PROGRAM TestStationControl
VAR
	(* These timers are used to imitate the moving time in the visualization*)
	T_Mat_Check: TIME := TIME#2S0MS;
	T1: TIME := TIME#2S0MS;
	T_liftDown: TIME := TIME#2S0MS;
	T_H_meas: TIME := TIME#2S0MS;
	T_MatPush: TIME := TIME#1S0MS;
	TON_Mat_Check: TON;
	TON_MatPush: TON;
	TON_MatPush2: TON;
	TON_Lift: TON;
	TON1: TON;
	TON_0: TON;
	TON_1: TON;
	TON_2: TON;
	TON_H_Meas: TON;
	TON_Lift2: TON;
	TON_reset: TON;
	
	(* These are just used to maintain the sequence or flow*)
	next2: BOOL;
	next3: BOOL;
	next4: BOOL;
END_VAR
VAR // added by the converter: edge detectors and wires of the graphical bodies
    _w1, _w2, _w3, _w4, _w5, _w6, _w7 : BOOL;
END_VAR

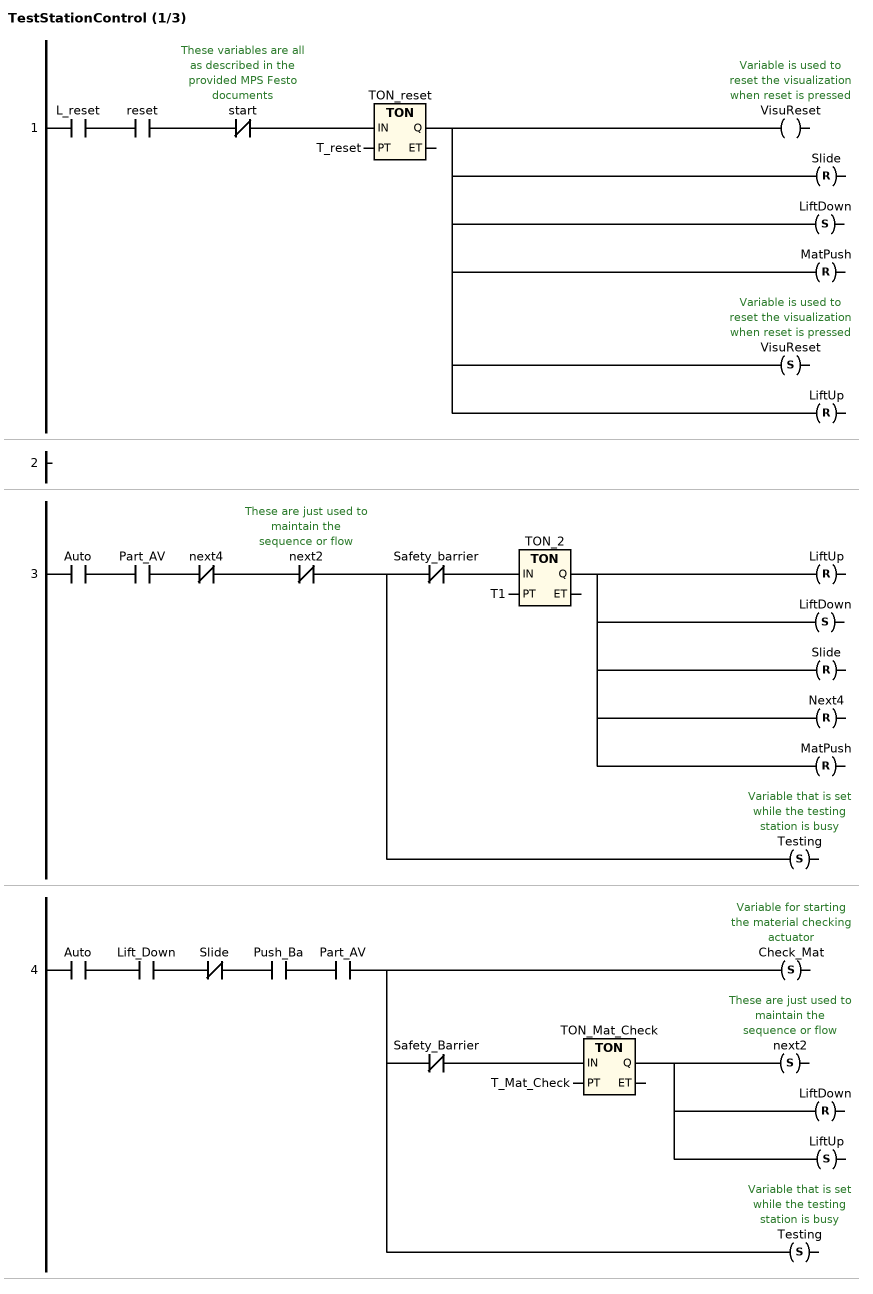
// NETWORK 1
//   start: These variables are all as described in the provided MPS Festo documents
//   T_reset: time to imitate reset value
//   VisuReset: Variable is used to reset the visualization when reset is pressed
TON_reset(IN := L_reset AND reset AND NOT start, PT := T_reset); // TON
VisuReset := TON_reset.Q;
Slide R= TON_reset.Q;
LiftDown S= TON_reset.Q;
MatPush R= TON_reset.Q;
VisuReset S= TON_reset.Q;
LiftUp R= TON_reset.Q;

// NETWORK 2

// NETWORK 3
//   next2: These are just used to maintain the sequence or flow
//   Testing: Variable that is set while the testing station is busy
_w1 := Auto AND Part_AV AND NOT next4 AND NOT next2;
TON_2(IN := _w1 AND NOT Safety_barrier, PT := T1); // TON
LiftUp R= TON_2.Q;
LiftDown S= TON_2.Q;
Slide R= TON_2.Q;
Next4 R= TON_2.Q;
MatPush R= TON_2.Q;
Testing S= _w1;

// NETWORK 4
//   Check_Mat: Variable for starting the material checking actuator
//   T_Mat_Check: These timers are used to imitate the moving time in the visualization
//   next2: These are just used to maintain the sequence or flow
//   Testing: Variable that is set while the testing station is busy
_w2 := Auto AND Lift_Down AND NOT Slide AND Push_Ba AND Part_AV;
Check_Mat S= _w2;
TON_Mat_Check(IN := _w2 AND NOT Safety_Barrier, PT := T_Mat_Check); // TON
next2 S= TON_Mat_Check.Q;
LiftDown R= TON_Mat_Check.Q;
LiftUp S= TON_Mat_Check.Q;
Testing S= _w2;

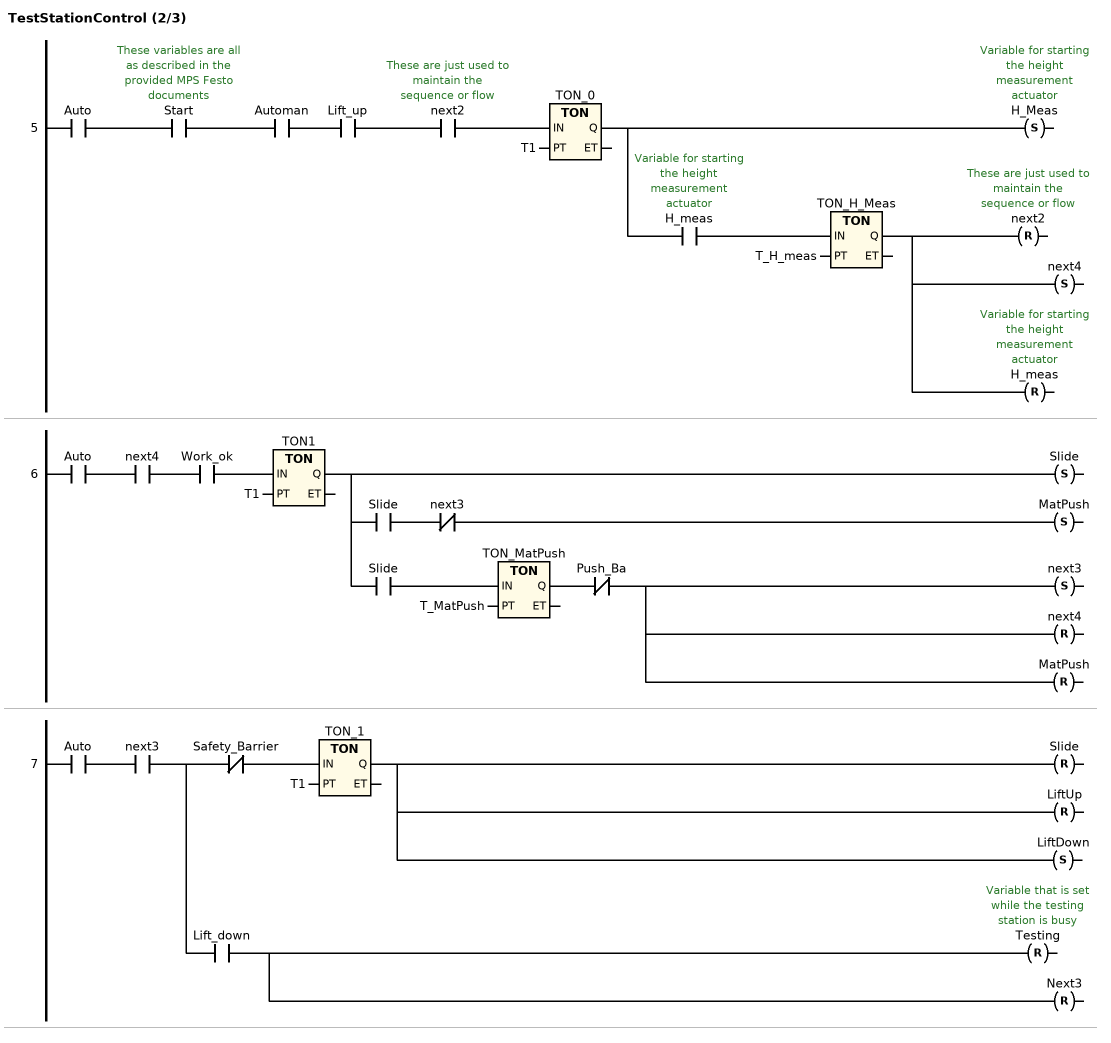
// NETWORK 5
//   Start: These variables are all as described in the provided MPS Festo documents
//   next2: These are just used to maintain the sequence or flow
//   H_Meas: Variable for starting the height measurement actuator
//   H_meas: Variable for starting the height measurement actuator
TON_0(IN := Auto AND Start AND Automan AND Lift_up AND next2, PT := T1); // TON
H_Meas S= TON_0.Q;
TON_H_Meas(IN := TON_0.Q AND H_meas, PT := T_H_meas); // TON
next2 R= TON_H_Meas.Q;
next4 S= TON_H_Meas.Q;
H_meas R= TON_H_Meas.Q;

// NETWORK 6
TON1(IN := Auto AND next4 AND Work_ok, PT := T1); // TON
Slide S= TON1.Q;
MatPush S= TON1.Q AND Slide AND NOT next3;
TON_MatPush(IN := TON1.Q AND Slide, PT := T_MatPush); // TON
_w3 := TON_MatPush.Q AND NOT Push_Ba;
next3 S= _w3;
next4 R= _w3;
MatPush R= _w3;

// NETWORK 7
//   Testing: Variable that is set while the testing station is busy
_w4 := Auto AND next3;
TON_1(IN := _w4 AND NOT Safety_Barrier, PT := T1); // TON
Slide R= TON_1.Q;
LiftUp R= TON_1.Q;
LiftDown S= TON_1.Q;
_w5 := _w4 AND Lift_down;
Testing R= _w5;
Next3 R= _w5;

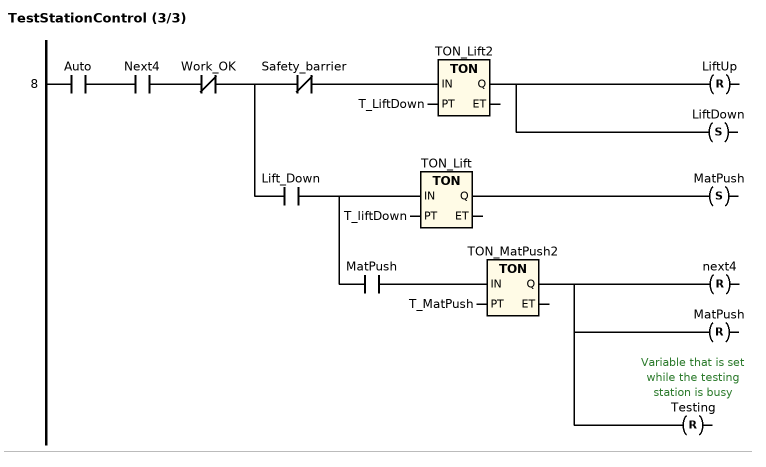
// NETWORK 8
//   Testing: Variable that is set while the testing station is busy
_w6 := Auto AND Next4 AND NOT Work_OK;
TON_Lift2(IN := _w6 AND NOT Safety_barrier, PT := T_LiftDown); // TON
LiftUp R= TON_Lift2.Q;
LiftDown S= TON_Lift2.Q;
_w7 := _w6 AND Lift_Down;
TON_Lift(IN := _w7, PT := T_liftDown); // TON
MatPush S= TON_Lift.Q;
TON_MatPush2(IN := _w7 AND MatPush, PT := T_MatPush); // TON
next4 R= TON_MatPush2.Q;
MatPush R= TON_MatPush2.Q;
Testing R= TON_MatPush2.Q;

END_PROGRAM

(* stored: Version 1.1.0.1, ProductVersion 3.1.4018.5
   POU TestStationControl: Id {270aeed6-7d97-4eb4-9d79-880ce9abfcf5}, SpecialFunc None *)
